// TIA Portal V18 export
FUNCTION "Operator message1" : Void   // FC29, LAD
{ S7_Optimized_Access := 'TRUE' }
VERSION : 0.1
// stored: AutoNumber true, IsIECCheckEnabled false, SetENOAutomatically false, UDAEnableTagReadback false
BEGIN

REGION Network 1
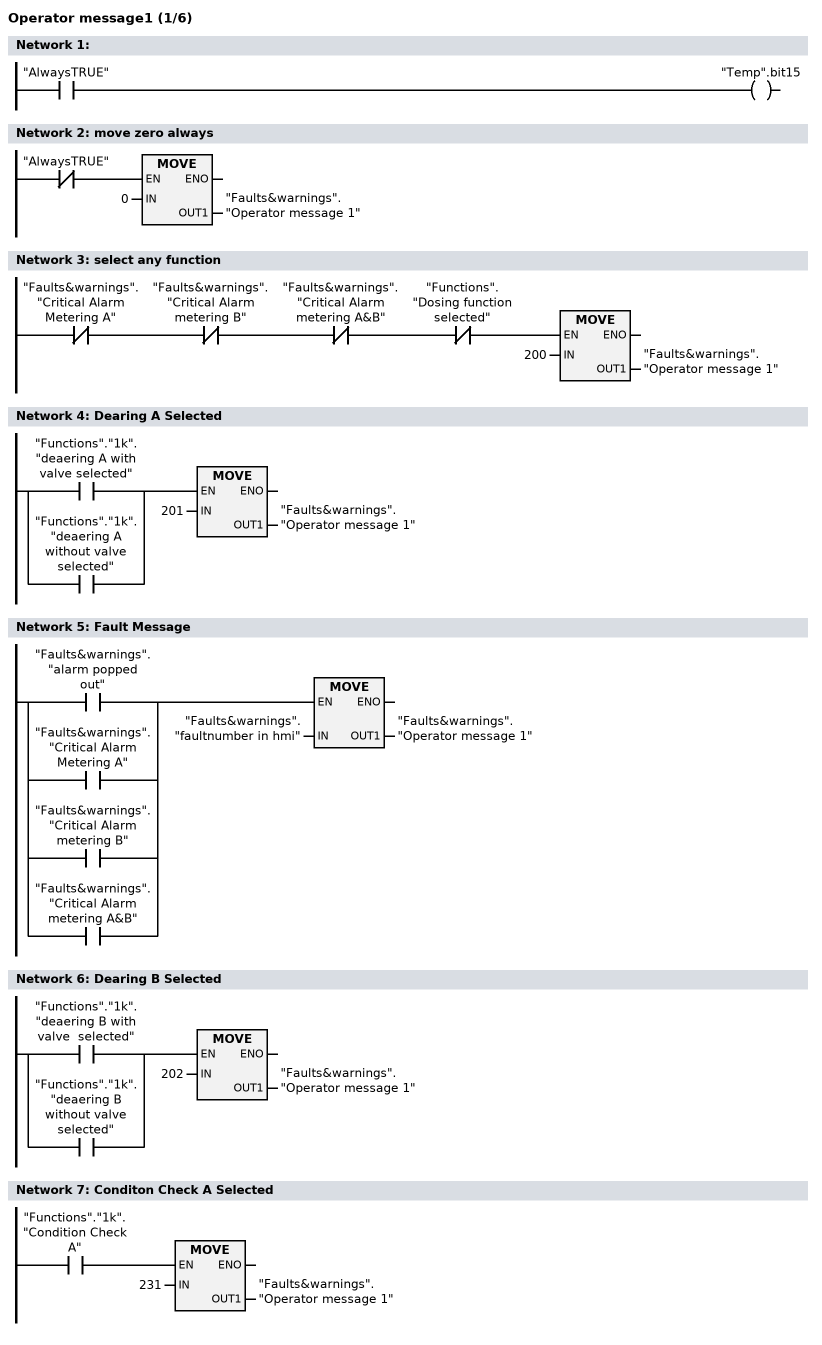
   RUNG wire#powerrail
      Contact( "AlwaysTRUE" )
      Coil( "Temp".bit15 )
   END_RUNG
   // the same network as SCL:
   "Temp".bit15 := "AlwaysTRUE";
END_REGION

REGION Network 2: move zero always
   RUNG wire#powerrail
      I_Contact( "AlwaysTRUE" )
      Move(in := 0, out1 => "Faults&warnings"."Operator message 1")
   END_RUNG
   // the same network as SCL:
   IF NOT "AlwaysTRUE" THEN "Faults&warnings"."Operator message 1" := 0; END_IF;
END_REGION

REGION Network 3: select any function
   RUNG wire#powerrail
      I_Contact( "Faults&warnings"."Critical Alarm Metering A" )
      I_Contact( "Faults&warnings"."Critical Alarm metering B" )
      I_Contact( "Faults&warnings"."Critical Alarm metering A&B" )
      I_Contact( "Functions"."Dosing function selected" )
      Move(in := 200, out1 => "Faults&warnings"."Operator message 1")
   END_RUNG
   // the same network as SCL:
   IF NOT "Faults&warnings"."Critical Alarm Metering A" AND NOT "Faults&warnings"."Critical Alarm metering B" AND NOT "Faults&warnings"."Critical Alarm metering A&B" AND NOT "Functions"."Dosing function selected" THEN
       "Faults&warnings"."Operator message 1" := 200;
   END_IF;
END_REGION

REGION Network 4: Dearing A Selected
   RUNG wire#powerrail
      Contact( "Functions"."1k"."deaering A with valve selected" )
      wire#w1
      Move(in := 201, out1 => "Faults&warnings"."Operator message 1")
   END_RUNG
   RUNG wire#powerrail
      Contact( "Functions"."1k"."deaering A without valve selected" )
   END_RUNG wire#w1
   // the same network as SCL:
   IF "Functions"."1k"."deaering A with valve selected" OR "Functions"."1k"."deaering A without valve selected" THEN
       "Faults&warnings"."Operator message 1" := 201;
   END_IF;
END_REGION

REGION Network 5: Fault Message
   RUNG wire#powerrail
      Contact( "Faults&warnings"."alarm popped out" )
      wire#w1
      Move(in := "Faults&warnings"."faultnumber in hmi", out1 => "Faults&warnings"."Operator message 1")
   END_RUNG
   RUNG wire#powerrail
      Contact( "Faults&warnings"."Critical Alarm Metering A" )
   END_RUNG wire#w1
   RUNG wire#powerrail
      Contact( "Faults&warnings"."Critical Alarm metering B" )
   END_RUNG wire#w1
   RUNG wire#powerrail
      Contact( "Faults&warnings"."Critical Alarm metering A&B" )
   END_RUNG wire#w1
   // the same network as SCL:
   IF "Faults&warnings"."alarm popped out" OR "Faults&warnings"."Critical Alarm Metering A" OR "Faults&warnings"."Critical Alarm metering B" OR "Faults&warnings"."Critical Alarm metering A&B" THEN
       "Faults&warnings"."Operator message 1" := "Faults&warnings"."faultnumber in hmi";
   END_IF;
END_REGION

REGION Network 6: Dearing B Selected
   RUNG wire#powerrail
      Contact( "Functions"."1k"."deaering B with valve  selected" )
      wire#w1
      Move(in := 202, out1 => "Faults&warnings"."Operator message 1")
   END_RUNG
   RUNG wire#powerrail
      Contact( "Functions"."1k"."deaering B without valve  selected" )
   END_RUNG wire#w1
   // the same network as SCL:
   IF "Functions"."1k"."deaering B with valve  selected" OR "Functions"."1k"."deaering B without valve  selected" THEN
       "Faults&warnings"."Operator message 1" := 202;
   END_IF;
END_REGION

REGION Network 7: Conditon Check A Selected
   RUNG wire#powerrail
      Contact( "Functions"."1k"."Condition Check A" )
      Move(in := 231, out1 => "Faults&warnings"."Operator message 1")
   END_RUNG
   // the same network as SCL:
   IF "Functions"."1k"."Condition Check A" THEN "Faults&warnings"."Operator message 1" := 231; END_IF;
END_REGION

REGION Network 8: Conditon Check B Selected
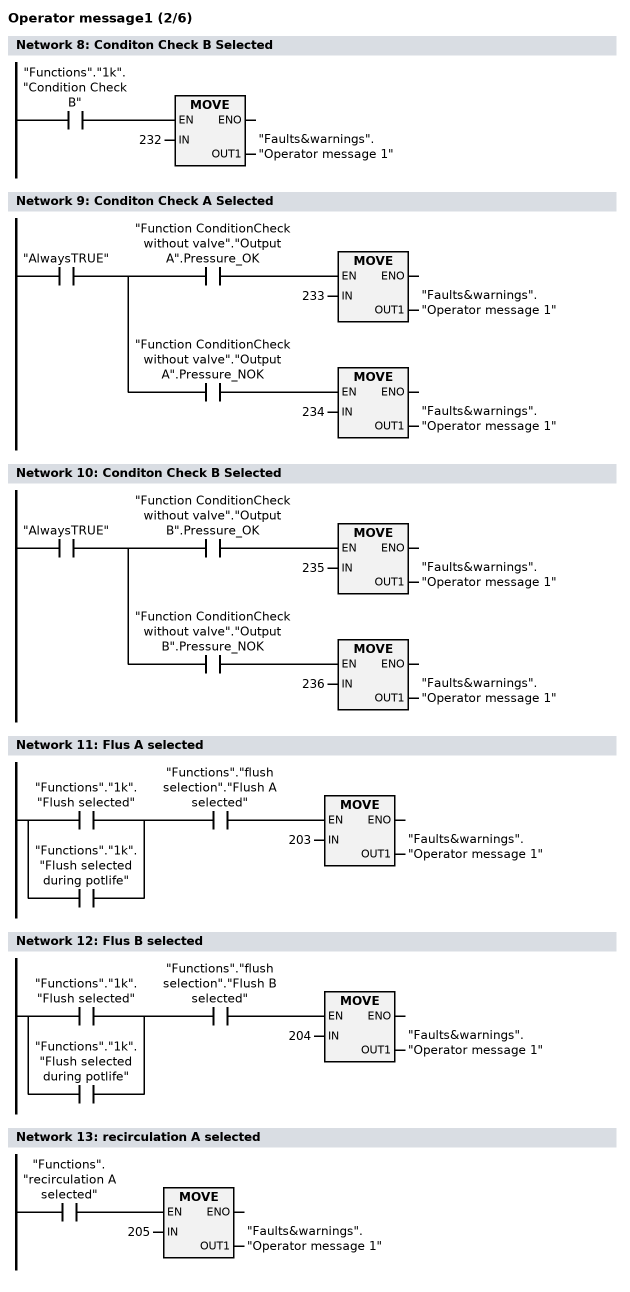
   RUNG wire#powerrail
      Contact( "Functions"."1k"."Condition Check B" )
      Move(in := 232, out1 => "Faults&warnings"."Operator message 1")
   END_RUNG
   // the same network as SCL:
   IF "Functions"."1k"."Condition Check B" THEN "Faults&warnings"."Operator message 1" := 232; END_IF;
END_REGION

REGION Network 9: Conditon Check A Selected
   RUNG wire#powerrail
      Contact( "AlwaysTRUE" )
      wire#w1
      Contact( "Function ConditionCheck without valve"."Output A".Pressure_OK )
      Move(in := 233, out1 => "Faults&warnings"."Operator message 1")
   END_RUNG
   RUNG wire#w1
      Contact( "Function ConditionCheck without valve"."Output A".Pressure_NOK )
      Move(in := 234, out1 => "Faults&warnings"."Operator message 1")
   END_RUNG
   // the same network as SCL:
   IF "AlwaysTRUE" AND "Function ConditionCheck without valve"."Output A".Pressure_OK THEN
       "Faults&warnings"."Operator message 1" := 233;
   END_IF;
   IF "AlwaysTRUE" AND "Function ConditionCheck without valve"."Output A".Pressure_NOK THEN
       "Faults&warnings"."Operator message 1" := 234;
   END_IF;
END_REGION

REGION Network 10: Conditon Check B Selected
   RUNG wire#powerrail
      Contact( "AlwaysTRUE" )
      wire#w1
      Contact( "Function ConditionCheck without valve"."Output B".Pressure_OK )
      Move(in := 235, out1 => "Faults&warnings"."Operator message 1")
   END_RUNG
   RUNG wire#w1
      Contact( "Function ConditionCheck without valve"."Output B".Pressure_NOK )
      Move(in := 236, out1 => "Faults&warnings"."Operator message 1")
   END_RUNG
   // the same network as SCL:
   IF "AlwaysTRUE" AND "Function ConditionCheck without valve"."Output B".Pressure_OK THEN
       "Faults&warnings"."Operator message 1" := 235;
   END_IF;
   IF "AlwaysTRUE" AND "Function ConditionCheck without valve"."Output B".Pressure_NOK THEN
       "Faults&warnings"."Operator message 1" := 236;
   END_IF;
END_REGION

REGION Network 11: Flus A selected
   RUNG wire#powerrail
      Contact( "Functions"."1k"."Flush selected" )
      wire#w1
      Contact( "Functions"."flush selection"."Flush A selected" )
      Move(in := 203, out1 => "Faults&warnings"."Operator message 1")
   END_RUNG
   RUNG wire#powerrail
      Contact( "Functions"."1k"."Flush selected during potlife" )
   END_RUNG wire#w1
   // the same network as SCL:
   IF ("Functions"."1k"."Flush selected" OR "Functions"."1k"."Flush selected during potlife") AND "Functions"."flush selection"."Flush A selected" THEN
       "Faults&warnings"."Operator message 1" := 203;
   END_IF;
END_REGION

REGION Network 12: Flus B selected
   RUNG wire#powerrail
      Contact( "Functions"."1k"."Flush selected" )
      wire#w1
      Contact( "Functions"."flush selection"."Flush B selected" )
      Move(in := 204, out1 => "Faults&warnings"."Operator message 1")
   END_RUNG
   RUNG wire#powerrail
      Contact( "Functions"."1k"."Flush selected during potlife" )
   END_RUNG wire#w1
   // the same network as SCL:
   IF ("Functions"."1k"."Flush selected" OR "Functions"."1k"."Flush selected during potlife") AND "Functions"."flush selection"."Flush B selected" THEN
       "Faults&warnings"."Operator message 1" := 204;
   END_IF;
END_REGION

REGION Network 13: recirculation A selected
   RUNG wire#powerrail
      Contact( "Functions"."recirculation A selected" )
      Move(in := 205, out1 => "Faults&warnings"."Operator message 1")
   END_RUNG
   // the same network as SCL:
   IF "Functions"."recirculation A selected" THEN "Faults&warnings"."Operator message 1" := 205; END_IF;
END_REGION

REGION Network 14: recirculation B selected
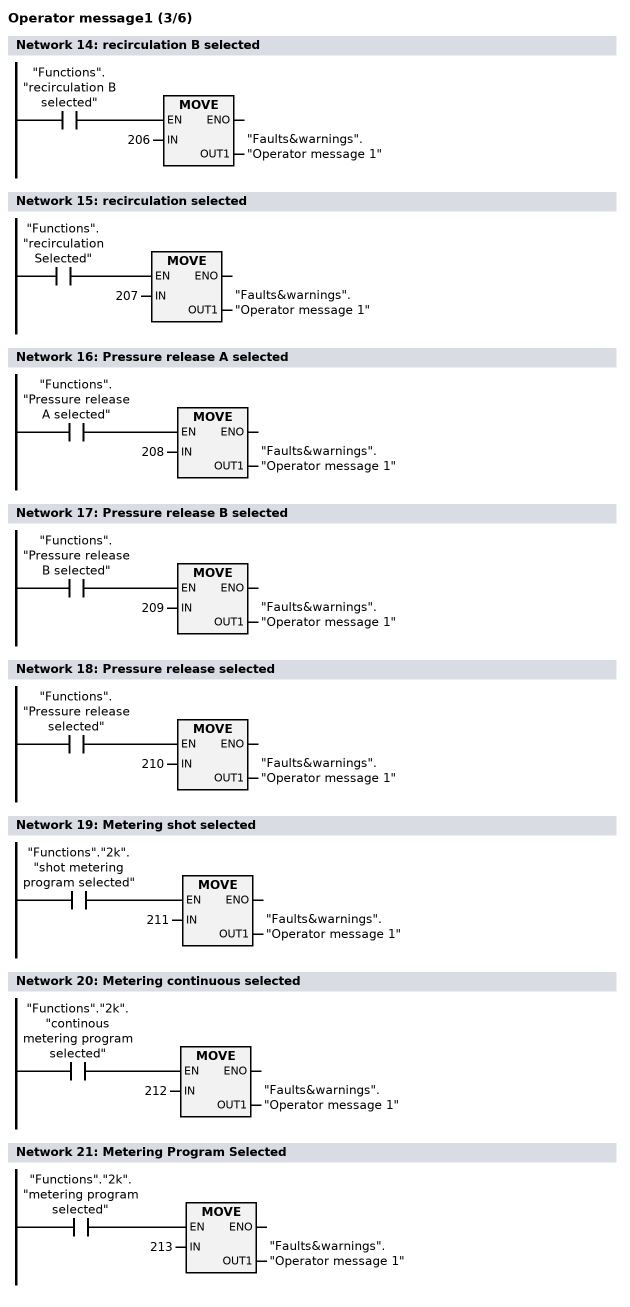
   RUNG wire#powerrail
      Contact( "Functions"."recirculation B selected" )
      Move(in := 206, out1 => "Faults&warnings"."Operator message 1")
   END_RUNG
   // the same network as SCL:
   IF "Functions"."recirculation B selected" THEN "Faults&warnings"."Operator message 1" := 206; END_IF;
END_REGION

REGION Network 15: recirculation selected
   RUNG wire#powerrail
      Contact( "Functions"."recirculation Selected" )
      Move(in := 207, out1 => "Faults&warnings"."Operator message 1")
   END_RUNG
   // the same network as SCL:
   IF "Functions"."recirculation Selected" THEN "Faults&warnings"."Operator message 1" := 207; END_IF;
END_REGION

REGION Network 16: Pressure release A selected
   RUNG wire#powerrail
      Contact( "Functions"."Pressure release A selected" )
      Move(in := 208, out1 => "Faults&warnings"."Operator message 1")
   END_RUNG
   // the same network as SCL:
   IF "Functions"."Pressure release A selected" THEN "Faults&warnings"."Operator message 1" := 208; END_IF;
END_REGION

REGION Network 17: Pressure release B selected
   RUNG wire#powerrail
      Contact( "Functions"."Pressure release B selected" )
      Move(in := 209, out1 => "Faults&warnings"."Operator message 1")
   END_RUNG
   // the same network as SCL:
   IF "Functions"."Pressure release B selected" THEN "Faults&warnings"."Operator message 1" := 209; END_IF;
END_REGION

REGION Network 18: Pressure release selected
   RUNG wire#powerrail
      Contact( "Functions"."Pressure release selected" )
      Move(in := 210, out1 => "Faults&warnings"."Operator message 1")
   END_RUNG
   // the same network as SCL:
   IF "Functions"."Pressure release selected" THEN "Faults&warnings"."Operator message 1" := 210; END_IF;
END_REGION

REGION Network 19: Metering shot selected
   RUNG wire#powerrail
      Contact( "Functions"."2k"."shot metering program selected" )
      Move(in := 211, out1 => "Faults&warnings"."Operator message 1")
   END_RUNG
   // the same network as SCL:
   IF "Functions"."2k"."shot metering program selected" THEN
       "Faults&warnings"."Operator message 1" := 211;
   END_IF;
END_REGION

REGION Network 20: Metering continuous selected
   RUNG wire#powerrail
      Contact( "Functions"."2k"."continous metering program selected" )
      Move(in := 212, out1 => "Faults&warnings"."Operator message 1")
   END_RUNG
   // the same network as SCL:
   IF "Functions"."2k"."continous metering program selected" THEN
       "Faults&warnings"."Operator message 1" := 212;
   END_IF;
END_REGION

REGION Network 21: Metering Program Selected
   RUNG wire#powerrail
      Contact( "Functions"."2k"."metering program selected" )
      Move(in := 213, out1 => "Faults&warnings"."Operator message 1")
   END_RUNG
   // the same network as SCL:
   IF "Functions"."2k"."metering program selected" THEN
       "Faults&warnings"."Operator message 1" := 213;
   END_IF;
END_REGION

REGION Network 22: Pre run Program Selected
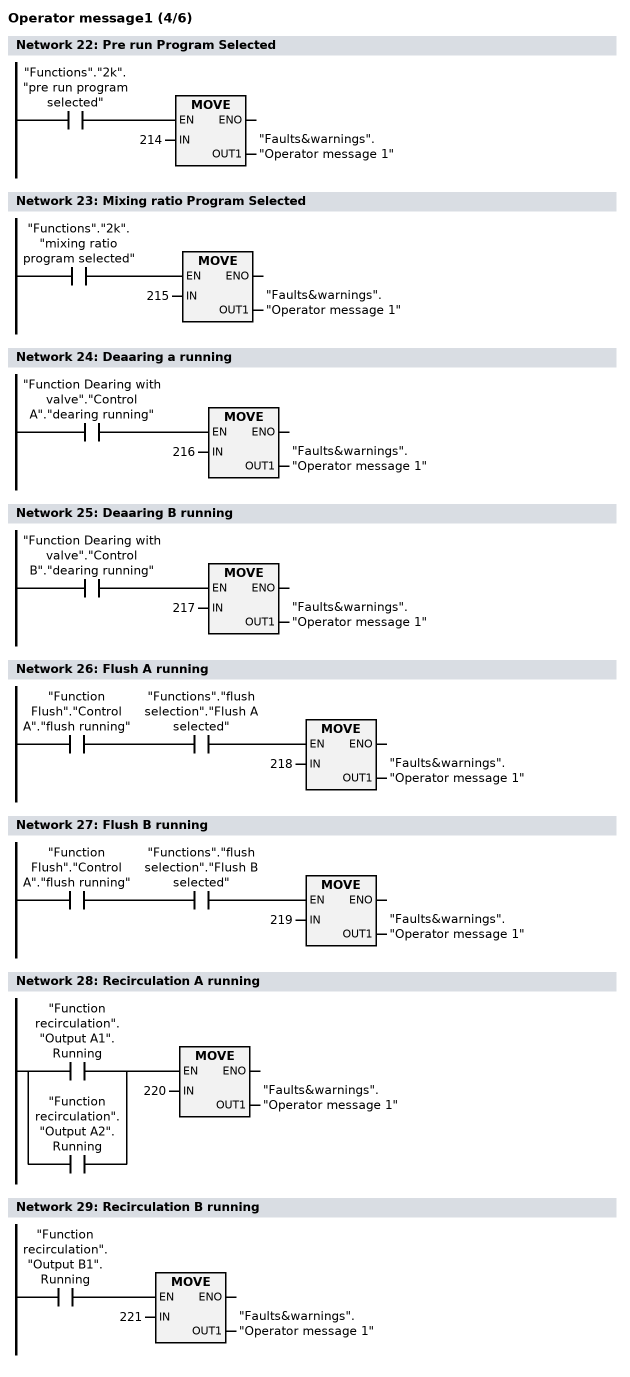
   RUNG wire#powerrail
      Contact( "Functions"."2k"."pre run program selected" )
      Move(in := 214, out1 => "Faults&warnings"."Operator message 1")
   END_RUNG
   // the same network as SCL:
   IF "Functions"."2k"."pre run program selected" THEN "Faults&warnings"."Operator message 1" := 214; END_IF;
END_REGION

REGION Network 23: Mixing ratio Program Selected
   RUNG wire#powerrail
      Contact( "Functions"."2k"."mixing ratio program selected" )
      Move(in := 215, out1 => "Faults&warnings"."Operator message 1")
   END_RUNG
   // the same network as SCL:
   IF "Functions"."2k"."mixing ratio program selected" THEN
       "Faults&warnings"."Operator message 1" := 215;
   END_IF;
END_REGION

REGION Network 24: Deaaring a running
   RUNG wire#powerrail
      Contact( "Function Dearing with valve"."Control A"."dearing running" )
      Move(in := 216, out1 => "Faults&warnings"."Operator message 1")
   END_RUNG
   // the same network as SCL:
   IF "Function Dearing with valve"."Control A"."dearing running" THEN
       "Faults&warnings"."Operator message 1" := 216;
   END_IF;
END_REGION

REGION Network 25: Deaaring B running
   RUNG wire#powerrail
      Contact( "Function Dearing with valve"."Control B"."dearing running" )
      Move(in := 217, out1 => "Faults&warnings"."Operator message 1")
   END_RUNG
   // the same network as SCL:
   IF "Function Dearing with valve"."Control B"."dearing running" THEN
       "Faults&warnings"."Operator message 1" := 217;
   END_IF;
END_REGION

REGION Network 26: Flush A running
   RUNG wire#powerrail
      Contact( "Function Flush"."Control A"."flush running" )
      Contact( "Functions"."flush selection"."Flush A selected" )
      Move(in := 218, out1 => "Faults&warnings"."Operator message 1")
   END_RUNG
   // the same network as SCL:
   IF "Function Flush"."Control A"."flush running" AND "Functions"."flush selection"."Flush A selected" THEN
       "Faults&warnings"."Operator message 1" := 218;
   END_IF;
END_REGION

REGION Network 27: Flush B running
   RUNG wire#powerrail
      Contact( "Function Flush"."Control A"."flush running" )
      Contact( "Functions"."flush selection"."Flush B selected" )
      Move(in := 219, out1 => "Faults&warnings"."Operator message 1")
   END_RUNG
   // the same network as SCL:
   IF "Function Flush"."Control A"."flush running" AND "Functions"."flush selection"."Flush B selected" THEN
       "Faults&warnings"."Operator message 1" := 219;
   END_IF;
END_REGION

REGION Network 28: Recirculation A running
   RUNG wire#powerrail
      Contact( "Function recirculation"."Output A1".Running )
      wire#w1
      Move(in := 220, out1 => "Faults&warnings"."Operator message 1")
   END_RUNG
   RUNG wire#powerrail
      Contact( "Function recirculation"."Output A2".Running )
   END_RUNG wire#w1
   // the same network as SCL:
   IF "Function recirculation"."Output A1".Running OR "Function recirculation"."Output A2".Running THEN
       "Faults&warnings"."Operator message 1" := 220;
   END_IF;
END_REGION

REGION Network 29: Recirculation B running
   RUNG wire#powerrail
      Contact( "Function recirculation"."Output B1".Running )
      Move(in := 221, out1 => "Faults&warnings"."Operator message 1")
   END_RUNG
   // the same network as SCL:
   IF "Function recirculation"."Output B1".Running THEN
       "Faults&warnings"."Operator message 1" := 221;
   END_IF;
END_REGION

REGION Network 30: Recirculation running
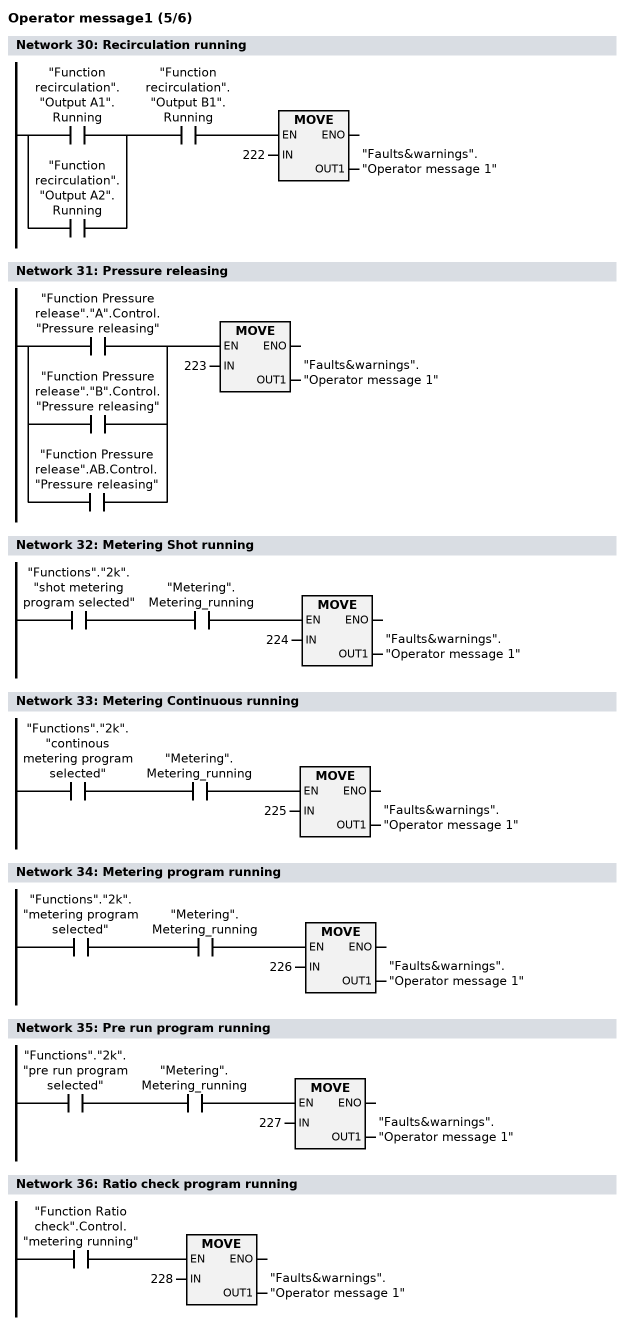
   RUNG wire#powerrail
      Contact( "Function recirculation"."Output A1".Running )
      wire#w1
      Contact( "Function recirculation"."Output B1".Running )
      Move(in := 222, out1 => "Faults&warnings"."Operator message 1")
   END_RUNG
   RUNG wire#powerrail
      Contact( "Function recirculation"."Output A2".Running )
   END_RUNG wire#w1
   // the same network as SCL:
   IF ("Function recirculation"."Output A1".Running OR "Function recirculation"."Output A2".Running) AND "Function recirculation"."Output B1".Running THEN
       "Faults&warnings"."Operator message 1" := 222;
   END_IF;
END_REGION

REGION Network 31: Pressure releasing
   RUNG wire#powerrail
      Contact( "Function Pressure release"."A".Control."Pressure releasing" )
      wire#w1
      Move(in := 223, out1 => "Faults&warnings"."Operator message 1")
   END_RUNG
   RUNG wire#powerrail
      Contact( "Function Pressure release"."B".Control."Pressure releasing" )
   END_RUNG wire#w1
   RUNG wire#powerrail
      Contact( "Function Pressure release".AB.Control."Pressure releasing" )
   END_RUNG wire#w1
   // the same network as SCL:
   IF "Function Pressure release"."A".Control."Pressure releasing" OR "Function Pressure release"."B".Control."Pressure releasing" OR "Function Pressure release".AB.Control."Pressure releasing" THEN
       "Faults&warnings"."Operator message 1" := 223;
   END_IF;
END_REGION

REGION Network 32: Metering Shot running
   RUNG wire#powerrail
      Contact( "Functions"."2k"."shot metering program selected" )
      Contact( "Metering".Metering_running )
      Move(in := 224, out1 => "Faults&warnings"."Operator message 1")
   END_RUNG
   // the same network as SCL:
   IF "Functions"."2k"."shot metering program selected" AND "Metering".Metering_running THEN
       "Faults&warnings"."Operator message 1" := 224;
   END_IF;
END_REGION

REGION Network 33: Metering Continuous running
   RUNG wire#powerrail
      Contact( "Functions"."2k"."continous metering program selected" )
      Contact( "Metering".Metering_running )
      Move(in := 225, out1 => "Faults&warnings"."Operator message 1")
   END_RUNG
   // the same network as SCL:
   IF "Functions"."2k"."continous metering program selected" AND "Metering".Metering_running THEN
       "Faults&warnings"."Operator message 1" := 225;
   END_IF;
END_REGION

REGION Network 34: Metering program running
   RUNG wire#powerrail
      Contact( "Functions"."2k"."metering program selected" )
      Contact( "Metering".Metering_running )
      Move(in := 226, out1 => "Faults&warnings"."Operator message 1")
   END_RUNG
   // the same network as SCL:
   IF "Functions"."2k"."metering program selected" AND "Metering".Metering_running THEN
       "Faults&warnings"."Operator message 1" := 226;
   END_IF;
END_REGION

REGION Network 35: Pre run program running
   RUNG wire#powerrail
      Contact( "Functions"."2k"."pre run program selected" )
      Contact( "Metering".Metering_running )
      Move(in := 227, out1 => "Faults&warnings"."Operator message 1")
   END_RUNG
   // the same network as SCL:
   IF "Functions"."2k"."pre run program selected" AND "Metering".Metering_running THEN
       "Faults&warnings"."Operator message 1" := 227;
   END_IF;
END_REGION

REGION Network 36: Ratio check program running
   RUNG wire#powerrail
      Contact( "Function Ratio check".Control."metering running" )
      Move(in := 228, out1 => "Faults&warnings"."Operator message 1")
   END_RUNG
   // the same network as SCL:
   IF "Function Ratio check".Control."metering running" THEN
       "Faults&warnings"."Operator message 1" := 228;
   END_IF;
END_REGION

REGION Network 37: Reneration program Selected
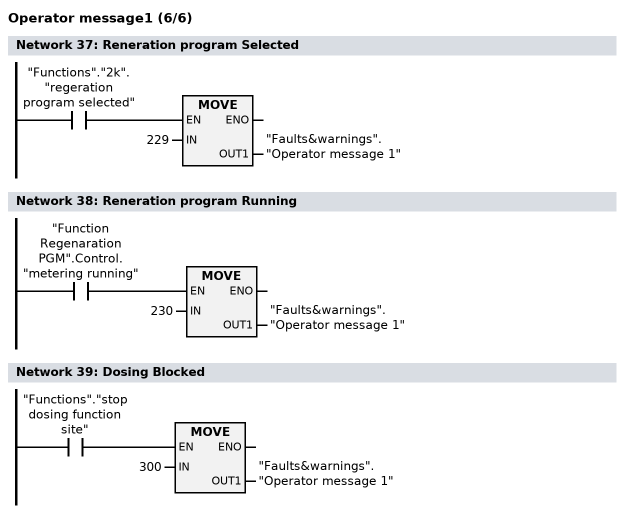
   RUNG wire#powerrail
      Contact( "Functions"."2k"."regeration program selected" )
      Move(in := 229, out1 => "Faults&warnings"."Operator message 1")
   END_RUNG
   // the same network as SCL:
   IF "Functions"."2k"."regeration program selected" THEN
       "Faults&warnings"."Operator message 1" := 229;
   END_IF;
END_REGION

REGION Network 38: Reneration program Running
   RUNG wire#powerrail
      Contact( "Function Regenaration PGM".Control."metering running" )
      Move(in := 230, out1 => "Faults&warnings"."Operator message 1")
   END_RUNG
   // the same network as SCL:
   IF "Function Regenaration PGM".Control."metering running" THEN
       "Faults&warnings"."Operator message 1" := 230;
   END_IF;
END_REGION

REGION Network 39: Dosing Blocked
   RUNG wire#powerrail
      Contact( "Functions"."stop dosing function site" )
      Move(in := 300, out1 => "Faults&warnings"."Operator message 1")
   END_RUNG
   // the same network as SCL:
   IF "Functions"."stop dosing function site" THEN "Faults&warnings"."Operator message 1" := 300; END_IF;
END_REGION

REGION Network 40 (SCL)
   // IF "Faults&warnings"."Status Nok"."Low level A1"  THEN
   //   "Faults&warnings"."Operator message 1" := 74;
   // END_IF;
   // IF "Faults&warnings"."Status Nok"."Low level B1" THEN
   //   "Faults&warnings"."Operator message 1" := 75;
   // END_IF;
   // IF "Alarm_DB".input.alarm[21] THEN
   //   "Faults&warnings"."Operator message 1" := 76;
   // END_IF;
   // IF "Alarm_DB".input.alarm[20] THEN
   //     "Faults&warnings"."Operator message 1" := 77;
   // END_IF;

   // IF "Faults&warnings"."Status Nok"."Level Low Drum A1" THEN
   //   "Faults&warnings"."Operator message 1" := 82;
   // END_IF;
   // IF "Faults&warnings"."Status Nok"."Level Low Drum B1" THEN
   //   "Faults&warnings"."Operator message 1" := 83;
   // END_IF;
   // IF "Faults&warnings"."Status Nok"."Level Low Drum A2" THEN
   //   "Faults&warnings"."Operator message 1" := 84;
   // END_IF;
   // IF "Faults&warnings"."Status Nok"."Level Low Drum B2" THEN
   //   "Faults&warnings"."Operator message 1" := 85;
   // END_IF;
   // IF "Faults&warnings"."Status Nok"."Level Empty Drum A1" THEN
   //   "Faults&warnings"."Operator message 1" := 86;
   // END_IF;
   // IF "Faults&warnings"."Status Nok"."Level Empty Drum B1" THEN
   //   "Faults&warnings"."Operator message 1" := 87;
   // END_IF;
   // IF "Faults&warnings"."Status Nok"."Level Empty Drum A2" THEN
   //   "Faults&warnings"."Operator message 1" := 88;
   // END_IF;
   // IF "Faults&warnings"."Status Nok"."Level Empty Drum B2" THEN
   //   "Faults&warnings"."Operator message 1" := 89;
   // END_IF;
END_REGION
END_FUNCTION
